{attribute 'qualified_only'}
VAR_GLOBAL
	N_MAX_POINTS : UINT := 10;
END_VAR

(* stored: Version 1.1.0.1, ProductVersion 3.1.4024.12
   GVL GVL_Interpolation: Id {c46a5d0f-179f-4848-ba20-fc2b88391dfd} *)
